(* IEC 61131-3 sources: acq-iii/Firmware PLC/ejemplo8, 1 file *)

(* ---- program.st ---- *)
PROGRAM program0
  VAR
    I1 AT %IX0.1 : BOOL;
    I2 AT %IX0.2 : BOOL;
    Q1 AT %QX0.1 : BOOL;
    OW1 AT %QW0 : UINT;
  END_VAR
  VAR
    MOVE5_ENO : BOOL;
    MOVE5_OUT : UINT;
  END_VAR

  MOVE5_OUT := MOVE(EN := I2 AND I1, IN := 0, ENO => MOVE5_ENO);
  Q1 := MOVE5_ENO;
  IF MOVE5_ENO THEN
      OW1 := MOVE5_OUT;
  END_IF;
END_PROGRAM

CONFIGURATION Config0

  RESOURCE Res0 ON PLC
    TASK task0(INTERVAL := T#20ms,PRIORITY := 0);
    PROGRAM instance0 WITH task0 : program0;
  END_RESOURCE
END_CONFIGURATION
